// TIA Portal V17 export
// export: Created 2023-02-14T02:49:16.0545723Z, ExportSetting WithDefaults, DisplayName Totally Integrated Automation Portal, DisplayVersion V17, DisplayName TIA Portal Openness, DisplayVersion V17, DisplayName TIA Portal Teamcenter Gateway, DisplayVersion V17, DisplayName TIA Portal Version Control Interface, DisplayVersion V17, DisplayName SINAMICS Startdrive Advanced, DisplayVersion V17, DisplayName SINAMICS Startdrive G130, G150, S120, S150, SINAMICS MV, S210, DisplayVersion V17, DisplayName SINAMICS Startdrive G110M, G120, G120C, G120D, G120P, G115D, DisplayVersion V17, DisplayName STEP 7 Professional, DisplayVersion V17, DisplayName STEP 7 Safety, DisplayVersion V17, DisplayName WinCC Professional, DisplayVersion V17
DATA_BLOCK "THE2_From_BT_To_Mixing"   // DB198
{ S7_Optimized_Access := 'FALSE' }
VERSION : 0.1
// stored: AutoNumber false, DBAccessibleFromOPCUA true, DBAccessibleFromWebserver true, IsOnlyStoredInLoadMemory false, IsWriteProtectedInAS false
   VAR RETAIN
      HeartBeat : Bool := TRUE;
      CIPEnable : Bool;
      LineProd_Open : Bool;
      LineCIP_Open : Bool;
      _free_4 : Bool;
      _free_5 : Bool;
      _free_6 : Bool;
      _free_7 : Bool;
      ProductRequest : Bool;
      _free_09 : Bool;
      _free_10 : Bool;
      _free_11 : Bool;
      _free_12 : Bool;
      _free_13 : Bool;
      _free_14 : Bool;
      _free_15 : Bool;
      _free_real2 : Real;
      _free_real6 : Real := 20000.0;
      _free_real10 : Real;
      _free_real14 : Real;
      _free_real18 : Real;
      _free_real22 : Real;
      _free_real26 : Real;
      _free_real30 : Real;
      FromTHE2Byte1 : Byte;
      FromTHE2Byte2 : Byte;
      FromTHE2Byte3 : Byte;
      FromTHE2Byte4 : Byte;
   END_VAR
BEGIN
END_DATA_BLOCK
